SUBAPPLICATION Uebung_020f (* DigitalInput_I1 auf DigitalOutput_Q1; E_PULSE; Impulsformend *)
  (* Standard: 61499-2 *)
  (* Version 1.0, 2023-10-23, franz *)
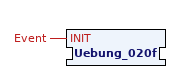
  EVENT_INPUT
    INIT;
  END_EVENT
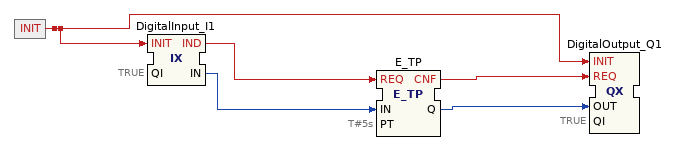
  FBS
    DigitalOutput_Q1 : QX(QI := TRUE);
    DigitalInput_I1 : IX(QI := TRUE);
    E_TP : E_TP(PT := T#5s);
  END_FBS
  EVENT_CONNECTIONS
    INIT TO DigitalInput_I1.INIT;
    INIT TO DigitalOutput_Q1.INIT;
    DigitalInput_I1.IND TO E_TP.REQ;
    E_TP.CNF TO DigitalOutput_Q1.REQ;
  END_CONNECTIONS
  DATA_CONNECTIONS
    DigitalInput_I1.IN TO E_TP.IN;
    E_TP.Q TO DigitalOutput_Q1.OUT;
  END_CONNECTIONS
END_SUBAPPLICATION
